FUNCTION_BLOCK MoverFactory EXTENDS Factory
VAR
	ptrMover : POINTER TO Mover;
	itfMover : ITF_Mover;
END_VAR

METHOD Create : ITF_Cyclic
VAR_INPUT
END_VAR
PtrMover := __NEW(Mover);
Create := ptrMover^;
IF __QUERYINTERFACE(Create,itfMover) THEN
	itfMover.SetMaxVelo(MaxVelocity := 4000.0);
END_IF
END_METHOD

END_FUNCTION_BLOCK

(* stored: Version 1.1.0.1, ProductVersion 3.1.4024.12
   POU MoverFactory: Id {5a1d286c-95ba-40eb-905b-4af4e4af9a92}, SpecialFunc None
   Method Create: Id {f5906e45-4f49-4852-a7ca-34487231f730} *)
